DATA_BLOCK "MotorSequence_Settings"
{ S7_Optimized_Access := 'FALSE' }
VERSION : 1.0
VAR
    StartInterval : Time := T#2s;
    StopInterval : Time := T#2s;
END_VAR
BEGIN
END_DATA_BLOCK
